Fanuc TP program (LS listing): test.ls

/PROG  TEST
/ATTR
OWNER		= MNEDITOR;
COMMENT		= "";
PROG_SIZE	= 269;
CREATE		= DATE 21-04-27  TIME 08:51:44;
MODIFIED	= DATE 21-10-19  TIME 04:04:22;
FILE_NAME	= ;
VERSION		= 0;
LINE_COUNT	= 11;
MEMORY_SIZE	= 597;
PROTECT		= READ_WRITE;
TCD:  STACK_SIZE	= 0,
      TASK_PRIORITY	= 50,
      TIME_SLICE	= 0,
      BUSY_LAMP_OFF	= 0,
      ABORT_REQUEST	= 0,
      PAUSE_REQUEST	= 0;
DEFAULT_GROUP	= 1,*,*,*,*;
CONTROL_CODE	= 00000000 00000000;
/APPL

AUTO_SINGULARITY_HEADER;
  ENABLE_SINGULARITY_AVOIDANCE   : TRUE;
/MN
   1:  UFRAME_NUM=9 ;
   2:  UTOOL_NUM=4 ;
   3:   ;
   4:J PR[29:LASER CURRENT] 100% FINE    ;
   5:   ;
   6:   ;
   7:   ;
   8:   ;
   9:   ;
  10:   ;
  11:   ;
/POS
/END
